# EPICS autosave request: iocBoot/ioc13pmac/auto_settings.req
file "CARS_8_motor_settings.req",         P=$(P)
